Fanuc TP program (LS listing): AAA_J_MOVE.LS

/PROG  AAA_J_MOVE
/ATTR
OWNER		= MNEDITOR;
COMMENT		= "";
PROG_SIZE	= 305;
CREATE		= DATE 31-01-10  TIME 13:34:10;
MODIFIED	= DATE 31-01-11  TIME 05:17:38;
FILE_NAME	= ;
VERSION		= 0;
LINE_COUNT	= 12;
MEMORY_SIZE	= 629;
PROTECT		= READ_WRITE;
TCD:  STACK_SIZE	= 0,
      TASK_PRIORITY	= 50,
      TIME_SLICE	= 0,
      BUSY_LAMP_OFF	= 0,
      ABORT_REQUEST	= 0,
      PAUSE_REQUEST	= 0;
DEFAULT_GROUP	= 1,*,*,*,*;
CONTROL_CODE	= 00000000 00000000;
/APPL
/APPL

AUTO_SINGULARITY_HEADER;
  ENABLE_SINGULARITY_AVOIDANCE   : TRUE;
/MN
   1:  UFRAME_NUM=1 ;
   2:  UTOOL_NUM=5 ;
   3:   ;
   4:J PR[270:TF5 Cal Mark Ctr] 50% FINE    ;
   5:   ;
   6:  PAUSE ;
   7:   ;
   8:  UTOOL_NUM=6 ;
   9:   ;
  10:  PR[271,3:TF6 Vision Ctr]=PR[270,3:TF5 Cal Mark Ctr]    ;
  11:   ;
  12:J PR[271:TF6 Vision Ctr] 25% FINE    ;
/POS
/END
